FUNCTION_BLOCK FbMission
VAR_INPUT
	xAutoRunning: BOOL;
	xMission1Start: BOOL;
	xMission1Done: BOOL;
	xMission2Start: BOOL;
	xMission2Done: BOOL;
END_VAR
VAR_OUTPUT
	xNoMission: BOOL;
	/// Busy 1 
	xMission1: BOOL;
	/// Busy 2 
	xMission2: BOOL;
END_VAR

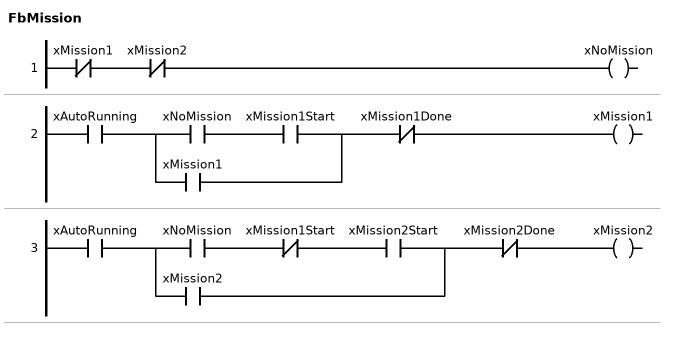
// NETWORK 1
xNoMission := NOT xMission1 AND NOT xMission2;

// NETWORK 2
xMission1 := xAutoRunning AND (xNoMission AND xMission1Start OR xMission1) AND NOT xMission1Done;

// NETWORK 3
xMission2 := xAutoRunning AND (xNoMission AND NOT xMission1Start AND xMission2Start OR xMission2) AND NOT xMission2Done;

END_FUNCTION_BLOCK

(* stored: Version 1.1.0.1, ProductVersion 3.1.4024.12
   POU FbMission: Id {ef40308d-36b2-42ba-87b7-49bcf334968e}, SpecialFunc None *)
